FUNCTION_BLOCK Valve (* Composite Function Block Type *)
  (* Standard: 61499-2 *)
  (* Version 0.0, 5/26/2016, Andrei, nxtControl GmbH, template *)
  PACKAGE Main;
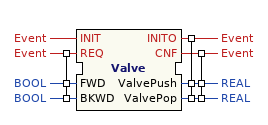
  EVENT_INPUT
    INIT; (* Initialization Request *)
    REQ WITH FWD, BKWD;
  END_EVENT
  EVENT_OUTPUT
    INITO WITH ValvePush, ValvePop; (* Initialization Confirm *)
    CNF WITH ValvePush, ValvePop;
  END_EVENT
  VAR_INPUT
    FWD : BOOL; (* Input event qualifier *)
    BKWD : BOOL;
  END_VAR
  VAR_OUTPUT
    ValvePush : REAL;
    ValvePop : REAL;
  END_VAR
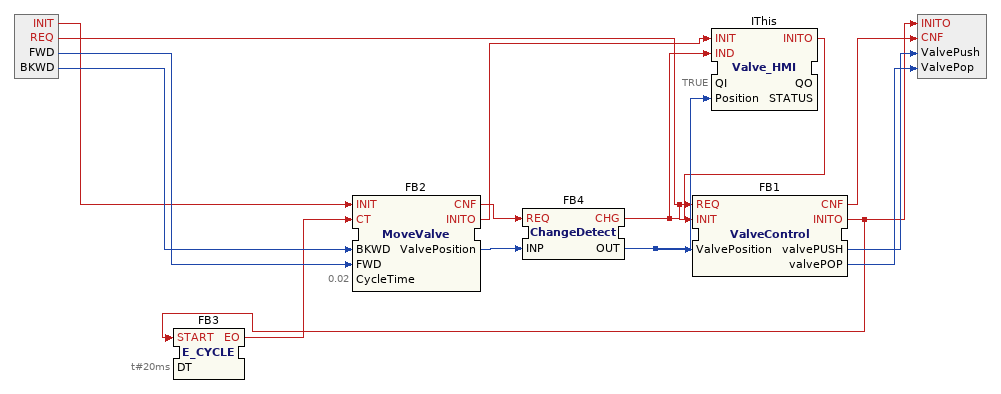
  FBS
    IThis : Valve_HMI(QI := TRUE);
    FB3 : E_CYCLE(DT := t#20ms);
    FB1 : ValveControl;
    FB2 : MoveValve(CycleTime := 0.02);
    FB4 : ChangeDetect;
  END_FBS
  EVENT_CONNECTIONS
    FB1.CNF TO CNF;
    INIT TO FB2.INIT;
    FB1.INITO TO INITO;
    FB3.EO TO FB2.CT;
    FB1.INITO TO FB3.START;
    REQ TO FB1.REQ;
    FB2.CNF TO FB4.REQ;
    FB4.CHG TO FB1.REQ;
    FB2.INITO TO IThis.INIT;
    FB4.CHG TO IThis.IND;
    IThis.INITO TO FB1.INIT;
  END_CONNECTIONS
  DATA_CONNECTIONS
    FB1.valvePUSH TO ValvePush;
    FB1.valvePOP TO ValvePop;
    BKWD TO FB2.BKWD;
    FWD TO FB2.FWD;
    FB2.ValvePosition TO FB4.INP;
    FB4.OUT TO FB1.ValvePosition;
    FB4.OUT TO IThis.Position;
  END_CONNECTIONS
END_FUNCTION_BLOCK
